{attribute 'qualified_only'}
VAR_GLOBAL
	MAX_SIZE : UINT := 4;
END_VAR

(* stored: Version 1.1.0.1, ProductVersion 3.1.4024.15
   GVL GVL: Id {ced9f844-e280-4f9b-9ea0-a88c969cbec8} *)
